// TIA Portal V16 export
// export: Created 2024-12-03T15:41:43.6797424Z, ExportSetting WithDefaults, DisplayName Totally Integrated Automation Portal, DisplayVersion V16 Update 6, DisplayName TIA Portal Version Control Interface, DisplayVersion V16 Update 2, DisplayName TIA Portal Openness, DisplayVersion V16 Update 6, DisplayName TIA Portal Teamcenter Gateway, DisplayVersion V16, DisplayName SINAMICS Startdrive Advanced, DisplayVersion V16 Update 5, DisplayName SINAMICS Startdrive G130, G150, S120, S150, SINAMICS MV, S210, DisplayVersion V16 Update 5, DisplayName SINAMICS Startdrive G110M, G120, G120C, G120D, G120P, G115D, DisplayVersion V16 Update 5, DisplayName STEP 7 Professional, DisplayVersion V16 Update 6, DisplayName STEP 7 Safety, DisplayVersion V16, DisplayName WinCC Advanced / Unified PC, DisplayVersion V16 Update 6
FUNCTION_BLOCK "Barcode_CONV_Wrapper"   // FB70, SCL
{ S7_Optimized_Access := 'TRUE' }
VERSION : 0.1
// stored: AutoNumber true, IsIECCheckEnabled false, IsRetainMemResEnabled false, MemoryReserve 100, SetENOAutomatically false, UDAEnableTagReadback false
   VAR_IN_OUT
      IO_Upstream : "Conveyor_UDT";
      IO_CurrentStream : "Conveyor_UDT";
      IO_Scanner_1 : "COGNEX_DATAMAN_LOGIC_UDT";
   END_VAR
   VAR
      scanner1 : "LC_Cognex_DataMan_FB";
      scan_1Done { S7_SetPoint := 'True'} : Bool;
   END_VAR
   VAR_TEMP
      T_ZoneInfo : "ZoneInfo";
      T_AppState : "ApplicationState_UDT";
      T_Tracking : "Tracking_Simple_UDT_1";
      T_NewResult : Bool;
   END_VAR
BEGIN
   #T_ZoneInfo := "ApplicationState_DB".ZoneNames[#IO_CurrentStream.Zone];
   #T_AppState := "ApplicationState_DB".Appstate[#T_ZoneInfo.AppStateIndex];

   #IO_Scanner_1.Settings.OffDelay := t#500ms;

   REGION Scanner_1

       #scanner1(IO_BarcodeScanner:=#IO_Scanner_1,
                IO_UpstreamConv:=#IO_Upstream,
                O_Tracking=> #T_Tracking,
                O_NewResult => #T_NewResult,
                IO_CurrentStream:=#IO_CurrentStream);

      IF #T_NewResult THEN
          #scan_1Done := 1;
      END_IF;

   END_REGION

   REGION COPY DATA

       #IO_CurrentStream.Status.ObjectOnConveyor := TRUE;

       IF #scan_1Done THEN
           #IO_CurrentStream.TrackingStat.Current.Barcode := #IO_Scanner_1.ReadingResult.Barcode;
           #IO_CurrentStream.TrackingCmd.InductNewTracking := true;
           #IO_CurrentStream.TrackingCmd.NewTrackingId := #IO_CurrentStream.TrackingStat.Current;
       END_IF;

   END_REGION

   REGION ACCUMULATE CURRENT STREAM 

       IF #IO_Scanner_1.Cmd.ScanAuto THEN
           #IO_CurrentStream.Cmd.Accumulate.Acc_Scan_1 := TRUE;
       END_IF;

       IF #scan_1Done THEN
           #scan_1Done := 0;
           #IO_CurrentStream.Cmd.Accumulate.Acc_Scan_1 := FALSE;
       END_IF;

   END_REGION
END_FUNCTION_BLOCK
